Universal Robots PolyScope program: rear_table_pickup_system.urp

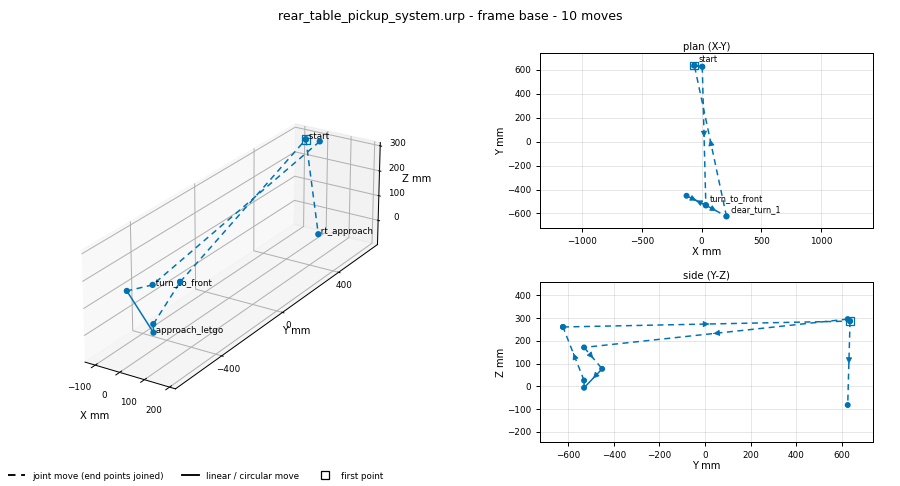
[picture p0: tool path of rear_table_pickup_system.urp in frame base, 10 of 12 moves have a stored position in this frame; points joined in program order, loops and branches not executed]
Program rear_table_pickup_system (installation=default directory=/programs/usbdisk_1/TVT19SPL createdIn=5.11.5.1010327 lastSavedIn=5.11.5.1010327 robotSerialNumber=20195600355)
Calibrated DH parameters: a=[0.000056, -0.161146, -0.252643, 0.000052, -0.000071, 0]; d=[0.181245, -342.672485, 975.135632, -632.288651, 0.119957, 0.115765]; alpha=[1.571164, 0.001314, -0.000405, 1.570615, -1.570559, 0]; deltaTheta=[0, -1.227166, 0.434415, 0.792759, -0.000001, 0]
BeforeStart
  URCap Gripper Activate (Robotiq_Grippers, Robotiq Inc.) dataModel(ResetAndActivateKey=false)
  URCap Gripper (Robotiq_Grippers, Robotiq Inc.) dataModel(position=0.0, force=100.0, speed=100.0, positionInDouble=0.0, forceInDouble=100.0, speedInDouble=100.0, slaveIds=[9], blocking=true)
Robot Program (runOnlyOnce=false)
  MoveJ speed 60 deg/s, acceleration 80 deg/s^2 (useActiveTCP=true) feature=Base
    Waypoint start: TCP in base x=-60.611 y=637.396 z=286.894 mm, rx=-0.4404 ry=-3.0971 rz=0.0094 rad; joints [259.31, -72.353, 84.496, -101.753, -89.31, 185.471] deg; TCP offset x=0 y=0 z=158.01 mm, rx=0 ry=0 rz=0 rad
